(* IEC 61131-3 sources: crb-codesys/generation/scripts/repoeval/测量控件/PRG, 1 file *)

(* ---- PLC_PRG.st ---- *)
PROGRAM PLC_PRG
VAR
	Tank01 : Tank;
END_VAR

Tank01(stName:='Tank01',nMaxLevel:=99, nMinLevel:=0,nMaxTemp:=55, nMinTemp:=44);
